(* CODESYS project CtaDevIOMb750362_1.0.0.0.library
   Description: Io System Library für Wago Modbbus Koppler 750-362 der CTA
   Version: 1.0.0.0
   Title: CtaDevIOMb750362
   Author: SIS
   DocFormat: reStructuredText
   LanguageModelAttribute: qualified-access-only
   Placeholder: CtaDevIOMb750362
   CompiledLibraryCompatibilityVersion: CODESYS V3.5 SP16 Patch 3
   Company: CTA
   DefaultNamespace: CtaDevIOMb750362

Project tree, tasks and I/O mapping:
  libraries: Standard, 3.5.18.0 (System); VisuDialogs, * (System); CtaSysConfig, 2.0.0.0 (CTA); CtaAppReport, 2.0.0.0 (CTA); CtaAppBmk, 2.0.0.0 (CTA); CtaAppInfluxLog, 1.0.0.1 (CTA); SysCom, 3.5.17.0 (System); CtaAppModbus, 2.0.0.0 (CTA); CtaSysIO, 2.0.0.0 (CTA); CtaVisSymbols, 2.0.0.0 (CTA)
  40 Visualizations/
    visualisation DIA_MB750362
    PFC_SLOT/
      SLOT/
        visualisation VIS_SLOT
        visualisation VIS_SLOT_QUERY
      FC/
        visualisation VIS_FC
        visualisation VIS_FC_QUERY
      visualisation FC_SLOT
      visualisation FC_SLOT_QUERY
    visualisation IO_ManagerBusInfo
    visualisation VIS_DYN_FC_IO_BASE
  30 Program Organization Units/
    function block FB_MB750362_KOPPLER [ST]: proVISU_DIA_NAME, actReport, BUS_ERROR, SIM_IO_TYPE
    FC/
      function fcScaleOut0_20mA [ST]
      function FcCheckIsDigitalIO [ST]
      function fcScaleOut4_20mA [ST]
      function fcGetTypeOfWagoSlot [ST]
      function fcScaleIN0_20mA [ST]
      function fcScaleOut0_10V [ST]
      function fcScaleIN0_10V [ST]
      function fcScaleIN4_20mA [ST]
      function fcScalePT1000 [ST]
      function fcGetModulImage [ST]
      function fcGetTypeOfWagoSlotSim [ST]
      function FcGetDigitalIOSim [ST]
  00000000-0000-0000-0000-000000000000|D:\CoDeSys\LibrariesV3\trunk\Intern\CAA\CAA Template\3.4.0.0 draft\Placeholder.xml
  00000000-0000-0000-0000-000000000000|D:\CoDeSys\LibrariesV3\trunk\Intern\CAA\CAA Template\3.2.0.3 draft\Prefix.pdf
  00000000-0000-0000-0000-000000000000|D:\CoDeSys\LibrariesV3\trunk\Intern\CAA\CAA Template\3.5.2.0 draft\Placeholder.xml
  20 Structs/
    data type scSlotInfo
    data type enModuleType
  50 Images/
    image pool WAGO_MB_IO_TERMINALS
  10 Documenation/
    global variables VersionHistory
    global variables readMe
  21 Interface/
  11 Library Parameter/
    global variables Parameter
  12 Konstanten/
  60 Textlisten/
    text list txtModulType
    text list txtWarning
    text list txtError
    text list txtPhysicalUnit
    text list txtInfo
  13 Globale Variablen/
    global variables GVL_TEXTLIST
  text list GlobalTextList
  5ce3da45-db07-42e7-a21c-a00fff4ed8f6|S:\_Temporär_SIS\CtaCodesysLibrary\01_Library\CtaSysIO\04_Image\0750_400.bmp
  5ce3da45-db07-42e7-a21c-a00fff4ed8f6|S:\_Temporär_SIS\CtaCodesysLibrary\01_Library\CtaSysIO\04_Image\0750_432.bmp
  5ce3da45-db07-42e7-a21c-a00fff4ed8f6|S:\_Temporär_SIS\CtaCodesysLibrary\01_Library\CtaSysIO\04_Image\0750_451.bmp
  5ce3da45-db07-42e7-a21c-a00fff4ed8f6|S:\_Temporär_SIS\CtaCodesysLibrary\01_Library\CtaSysIO\04_Image\0750_455.bmp
  5ce3da45-db07-42e7-a21c-a00fff4ed8f6|S:\_Temporär_SIS\CtaCodesysLibrary\01_Library\CtaSysIO\04_Image\0750_459.bmp
  5ce3da45-db07-42e7-a21c-a00fff4ed8f6|S:\_Temporär_SIS\CtaCodesysLibrary\01_Library\CtaSysIO\04_Image\0750_466.bmp
  5ce3da45-db07-42e7-a21c-a00fff4ed8f6|S:\_Temporär_SIS\CtaCodesysLibrary\01_Library\CtaSysIO\04_Image\0750_515.bmp
  5ce3da45-db07-42e7-a21c-a00fff4ed8f6|S:\_Temporär_SIS\CtaCodesysLibrary\01_Library\CtaSysIO\04_Image\0750_597.bmp
  5ce3da45-db07-42e7-a21c-a00fff4ed8f6|\\cta.local\mue\Daten\200_Klima_Kälte\200_300_KK_CTA_Exklusiv_Elektro\01_Elektro\03_Software\00_CtaCodesysLibrary\01_Library\CtaDevIOMb750362\04_Image\0750_600.bmp
  5ce3da45-db07-42e7-a21c-a00fff4ed8f6|S:\_Temporär_SIS\CtaCodesysLibrary\01_Library\CtaSysIO\04_Image\0750_652.bmp
  5ce3da45-db07-42e7-a21c-a00fff4ed8f6|S:\_Temporär_SIS\CtaCodesysLibrary\01_Library\CtaSysIO\04_Image\0750_1405.bmp
  5ce3da45-db07-42e7-a21c-a00fff4ed8f6|S:\_Temporär_SIS\CtaCodesysLibrary\01_Library\CtaSysIO\04_Image\0750_1415.bmp
  5ce3da45-db07-42e7-a21c-a00fff4ed8f6|S:\_Temporär_SIS\CtaCodesysLibrary\01_Library\CtaSysIO\04_Image\0750_1504.bmp
  5ce3da45-db07-42e7-a21c-a00fff4ed8f6|P:\200_Klima_Kälte\200_300_KK_CTA_Exklusiv_Elektro\01_Elektro\03_Software\00_CtaCodesysLibrary\01_Library\CtaDevIOMb750362\04_Image\0750_362.png
  5ce3da45-db07-42e7-a21c-a00fff4ed8f6|\\cta.local\mue\Daten\200_Klima_Kälte\200_300_KK_CTA_Exklusiv_Elektro\01_Elektro\03_Software\00_CtaCodesysLibrary\01_Library\CtaDevIOMb750362\04_Image\0750_BLANK.bmp
  5ce3da45-db07-42e7-a21c-a00fff4ed8f6|S:\_Temporär_SIS\CtaCodesysLibrary\01_Library\CtaSysIO\04_Image\0750_555.bmp
*)

// 20 Structs/scSlotInfo
TYPE scSlotInfo :
	STRUCT
		uiOrderNr	:	UINT;
		xDigital	:	BOOL;
		xInput		:	BOOL;
		uiFirstData	:	UINT;
		uiLastData	:	UINT;
		byAnzIoSlot	:	BYTE;
		enModulType :	enModuleType;
	END_STRUCT
END_TYPE

// 20 Structs/enModuleType
{attribute 'qualified_only'}
{attribute 'strict'}
{attribute 'to_string'}
TYPE enModuleType :
(
	Unknown 		:= 0,
	Digital_IN		:= 1,
	Digital_OUT		:= 2,	
	DC_0_10V_OUT	:= 3,
	DC_4_20mA_OUT	:= 4,
	DC_0_10V_IN		:= 5,
	DC_4_20mA_IN	:= 6,
	OHM				:= 7,
    RS485			:= 8,
	DC_0_20mA_OUT	:= 9,
	TEMPERATUR		:= 10,
	FCMB750362		:= 99
);
END_TYPE

// 10 Documenation/VersionHistory
(* 

.. image:: ../../Images/CTA_Logo.jpg
   :align: right
   :width: 15% 

**Vorlage**   


============ =========== =========== ============================================
**Date**     **Version** **Author**  **Change**
------------ ----------- ----------- --------------------------------------------
04.03.2021   0.0.0.0     SIS         Vorlage erstellt

============ =========== =========== ============================================


*)
VAR_GLOBAL
    stInfo : STRING:= '0.0.0.0, Vorlage, CTA';
END_VAR

// 10 Documenation/readMe
(*

**ReadMe**
 
|	**Empfehlung**
|
|	Dokumentrieren Sie die Library für eine nachhaltige Entwicklung
|     
| *Beispiel*
| 
| Dies ist die Vorlage Library der CTA. Erstellen Sie ihre Library anhand dieser Vorlage.
*)

VAR_GLOBAL
    xReadMeDone              :   BOOL;
END_VAR

// 11 Library Parameter/Parameter
{attribute 'qualified_only'}
VAR_GLOBAL CONSTANT

END_VAR

// 13 Globale Variablen/GVL_TEXTLIST
{attribute 'qualified_only'}
VAR_GLOBAL CONSTANT
	stErrorTextlist		:	CtaAppReport.stReportTextList	:= 'CtaDevIOMb750362.txtError';
	stWarningTextlist	:	CtaAppReport.stReportTextList	:= 'CtaDevIOMb750362.txtWarning';
	stInfoTextlist		:	CtaAppReport.stReportTextList	:= 'CtaDevIOMb750362.txtInfo';
END_VAR

// 30 Program Organization Units/FB_MB750362_KOPPLER
FUNCTION_BLOCK FB_MB750362_KOPPLER EXTENDS CtaSysIO.FB_IO_DEVICE
VAR_INPUT
	ITF_CLIENT_IN		:	CtaAppModbus.ITF_CLIENT;
END_VAR
VAR_OUTPUT
	xAcknowledge		:	BOOL;
	xLockDown			:	BOOL;
END_VAR
VAR
	(* Data *)
	_wKbusReset			:	WORD;
	_wSoftWareReset		:	WORD;
	_ayDiagnose			:	ARRAY[0..0001]	OF WORD;
	_ayWatchDog			:	ARRAY[0..0010] 	OF WORD;
	_aySlotType			:	ARRAY[0..0255] 	OF WORD;
	_ayIOQuantity		:	ARRAY[0..0003] 	OF WORD;
	_ayAnalogInput		:	ARRAY[0..1020]	OF WORD;
	_ayAnalogOutput		:	ARRAY[0..1020]	OF WORD;
	_ayDigitalInput		:	ARRAY[0..0511]	OF BOOL;
	_ayDigitalOutput	:	ARRAY[0..0511]	OF BOOL;
	_aySlotInfo			:	ARRAY[0..0255]	OF scSlotInfo;	
	byAnzSlots			:	BYTE;
	(* Help Variable *)
	xTrigResetDevError	:	BOOL;
	xTrigResetSlotError	:	BOOL;
	xReset				:	BOOL;
	usiCase				:	USINT;
	diFor				:	DINT;
	diFor2				:	DINT;	
	diStartFor			:	DINT;
	diMaxCreatePerCycle	:	DINT	:= 50;	
	byAnzIoSlot			:	BYTE;
	uiNextAnalogInput	:	UINT;
	uiNextAnalogOutput	:	UINT;
	uiNextDigitalInput	:	UINT;
	uiNextDigitalOutput :	UINT;
	ITF_SLOT_TEMP		:	CtaSysIO.ITF_IO_SLOT;
	ITF_DI_TEMP			:	CtaSysIO.ITF_DI;
	ITF_DO_TEMP			:	CtaSysIO.ITF_DO;
	ITF_AI_TEMP			:	CtaSysIO.ITF_AI;
	ITF_AO_TEMP			:	CtaSysIO.ITF_AO;
	enType				:	CtaSysIO.enIOType;
	xTempAlUnterlauf	:	BOOL;
	xTempAlUeberlauf	:	BOOL;
	rTempPhysicalValue	:	REAL;
	tErrorDelayMb		:	TIME	:= T#20S;
	xBusError			:	BOOL;
	scReportNr			:	CtaAppReport.scReportNr;
	fbReportManager		:	CtaAppReport.fbReportManager;
	fbMbErrorReport		:	CtaAppReport.fbReporter;
	fbDevErrorReport	:	CtaAppReport.fbReporter;
	fbWarningReportHand	:	CtaAppReport.fbReporter;
	fbSlotMissmatch		:	CtaAppReport.fbReporter;
END_VAR;

SUPER^();
IF NOT SIMULATION_ENABLED THEN
	IF __QUERYINTERFACE(ITF_CLIENT_IN,ITF_CLIENT_IN) THEN
		xBusError := ITF_CLIENT_IN.ERROR;
		CASE usiCase OF 
			0:  (* Set Image *)
				IMAGE := '.WAGO_MB_IO_TERMINALS.0750_362';
				(* Read Watchdog State *)
				ITF_CLIENT_IN.CREATE_JOB(_byMbFunction := 04,_wMbAdress := 4102,_pData := ADR(_ayWatchDog[006])	,_wQuantity := 01);
				
				(* Reset K-Bus *)
				ITF_CLIENT_IN.CREATE_JOB(_byMbFunction := 06,_wMbAdress := 4139,_pData := ADR(_wKbusReset)		,_wQuantity := 01);
	
				(* Diagnose Info *)
				ITF_CLIENT_IN.CREATE_JOB(_byMbFunction := 04,_wMbAdress := 4128,_pData := ADR(_ayDiagnose[000])	,_wQuantity := 2);
				
				(* Next Step *)
				usiCase := usiCase + 1;
				
			1:	(* Wait *)
				IF ITF_CLIENT_IN.CONFIRM_ALL_JOBS_DONE THEN
					(* Next Step *)
					usiCase := usiCase + 1;
				END_IF;
				
			2:	(* Watchdog State evaluvation *)
				IF _ayWatchDog[06] = 0 THEN // Watchdog inaktive
					(* Set Watchdog Time *)
					_ayWatchDog[00]	:= 16#0032;	// Watchdog Time 5s
					ITF_CLIENT_IN.CREATE_JOB(_byMbFunction := 06,_wMbAdress := 4096,_pData := ADR(_ayWatchDog[000])	,_wQuantity := 01);
					(* Set Watchdog Reset Funktion *)
					_ayWatchDog[01]	:= 16#FFFF;	// Reset on FC1-FC16
					ITF_CLIENT_IN.CREATE_JOB(_byMbFunction := 06,_wMbAdress := 4097,_pData := ADR(_ayWatchDog[001])	,_wQuantity := 01);
					(* Remove Watchdog Stop Call *)
					ITF_CLIENT_IN.DESTROY_JOB(_byMbFunction := 06,_wMbAdress := 4104,_pData := ADR(_ayWatchDog[008])	,_wQuantity := 01);
					(* Remove K-Bus reset *)
					ITF_CLIENT_IN.DESTROY_JOB(_byMbFunction := 06,_wMbAdress := 4139,_pData := ADR(_wKbusReset)		,_wQuantity := 01);
					(* Remove Software reset *)
					ITF_CLIENT_IN.DESTROY_JOB(_byMbFunction := 06,_wMbAdress :=8256,_pData 	:=	 ADR(_wSoftWareReset),	_wQuantity	 :=	 1);
					(* Next Step after Watchdog Set *)
					usiCase := usiCase + 1;
				(* Stop Watchdog if allredy aktive *)
				ELSIF _ayWatchDog[06] = 1 OR _ayWatchDog[06] = 2 THEN // Watchdog aktive or Watchdog expired
					_ayWatchDog[08]	:= 16#AA55;	// Watchdog Stop
					ITF_CLIENT_IN.CREATE_JOB(_byMbFunction := 06,_wMbAdress := 4104,_pData := ADR(_ayWatchDog[008])	,_wQuantity := 01); 
				END_IF;
				
			3:	(* Wait *)
				IF ITF_CLIENT_IN.CONFIRM_ALL_JOBS_DONE THEN
					(* Next Step *)
					usiCase := usiCase + 1;
				END_IF;
				
			4: (* Check if Watchdog is Running *)
					(* Read Slots *)
					ITF_CLIENT_IN.CREATE_JOB(_byMbFunction 	:= 04,	_wMbAdress 	:= 8240,	_pData 	:=	 ADR(_aySlotType[000]),	_wQuantity	 :=	 65);
					ITF_CLIENT_IN.CREATE_JOB(_byMbFunction 	:= 04,	_wMbAdress 	:= 8241,	_pData 	:=	 ADR(_aySlotType[065]),	_wQuantity	 :=	 64);
					ITF_CLIENT_IN.CREATE_JOB(_byMbFunction 	:= 04,	_wMbAdress 	:= 8242,	_pData 	:=	 ADR(_aySlotType[129]),	_wQuantity	 :=	 64);
					ITF_CLIENT_IN.CREATE_JOB(_byMbFunction 	:= 04,	_wMbAdress 	:= 8243,	_pData 	:=	 ADR(_aySlotType[193]),	_wQuantity	 :=	 63);	
					
					(* Read Quantity of I/O *)                                          	       	  	                                  	   	
					ITF_CLIENT_IN.CREATE_JOB(_byMbFunction 	:= 04,	_wMbAdress 	:= 4130,	_pData 	:=	 ADR(_ayIOQuantity[0]),	_wQuantity	 :=	 04);	
				IF _ayWatchDog[06] = 1 THEN	
					(* Remove Watchdog Configs *)                                       	       	  	                                  	   	
					ITF_CLIENT_IN.DESTROY_JOB(_byMbFunction := 06,	_wMbAdress 	:= 4096,	_pData 	:=	 ADR(_ayWatchDog[000]),	_wQuantity	 :=	 01);
					ITF_CLIENT_IN.DESTROY_JOB(_byMbFunction := 06,	_wMbAdress 	:= 4097,	_pData 	:=	 ADR(_ayWatchDog[001]),	_wQuantity	 :=	 01);
					
					(* Next Step *)
					usiCase := usiCase + 1;                                             	       	  	                                       	
				END_IF;    
																														
			5:	(* Wait *)                                                              	       	  	                                       	
				IF ITF_CLIENT_IN.CONFIRM_ALL_JOBS_DONE THEN 
					(* Next Step *)                            	       	  	                                       	
					usiCase := usiCase + 1;                                             	       	  	                                       	
				END_IF;	
																															
			6: 	(* Delete Slot Jobs *)                                                  	       	  	                                       	
				ITF_CLIENT_IN.DESTROY_JOB(_byMbFunction 	:= 04,	_wMbAdress 	:= 8240,	_pData 	:=	 ADR(_aySlotType[000]),	_wQuantity	 :=	 65);
				ITF_CLIENT_IN.DESTROY_JOB(_byMbFunction 	:= 04,	_wMbAdress 	:= 8241,	_pData 	:=	 ADR(_aySlotType[065]),	_wQuantity	 :=	 64);
				ITF_CLIENT_IN.DESTROY_JOB(_byMbFunction 	:= 04,	_wMbAdress 	:= 8242,	_pData 	:=	 ADR(_aySlotType[129]),	_wQuantity	 :=	 64);
				ITF_CLIENT_IN.DESTROY_JOB(_byMbFunction 	:= 04,	_wMbAdress 	:= 8243,	_pData 	:=	 ADR(_aySlotType[193]),	_wQuantity	 :=	 63);	
				
				(* Delte Quantity of I/O *)                                             	       	  	                                  	   	
				ITF_CLIENT_IN.DESTROY_JOB(_byMbFunction 	:= 04,	_wMbAdress 	:= 4130,	_pData 	:=	 ADR(_ayIOQuantity[0]),	_wQuantity	 :=	 04);
				
				(* Add Read Analog Input Jobs as needed *)  
				IF (_ayIOQuantity[1] / 16) >= 001 THEN   // Quantity is Bit Orientet /16 = Dezimal                                           	       	  	                                  	   	
					ITF_CLIENT_IN.CREATE_JOB(_byMbFunction 		:= 04,	_wMbAdress 	:= 0000,	_pData 	:=	 ADR(_ayAnalogInput[000]),	_wQuantity	 :=	 MAX(1,MIN(085,(_ayIOQuantity[1] / 16) -000)));
				END_IF;
				IF (_ayIOQuantity[1] / 16) >= 085 THEN   // Quantity is Bit Orientet /16 = Dezimal 
					ITF_CLIENT_IN.CREATE_JOB(_byMbFunction 		:= 04,	_wMbAdress 	:= 0085,	_pData 	:=	 ADR(_ayAnalogInput[085]),	_wQuantity	 :=	 MAX(1,MIN(085,(_ayIOQuantity[1] / 16) -085)));
				END_IF;
				IF (_ayIOQuantity[1] / 16) >= 170 THEN   // Quantity is Bit Orientet /16 = Dezimal 
					ITF_CLIENT_IN.CREATE_JOB(_byMbFunction 		:= 04,	_wMbAdress 	:= 0170,	_pData 	:=	 ADR(_ayAnalogInput[170]),	_wQuantity	 :=	 MAX(1,MIN(086,(_ayIOQuantity[1] / 16) -170)));
				END_IF;
				IF (_ayIOQuantity[1] / 16) >= 256 THEN   // Quantity is Bit Orientet /16 = Dezimal 
					ITF_CLIENT_IN.CREATE_JOB(_byMbFunction 		:= 04,	_wMbAdress 	:=24576,	_pData 	:=	 ADR(_ayAnalogInput[256]),	_wQuantity	 :=	 MAX(1,MIN(120,(_ayIOQuantity[1] / 16) -256)));
				END_IF;
				IF (_ayIOQuantity[1] / 16) >= 376 THEN   // Quantity is Bit Orientet /16 = Dezimal 
					ITF_CLIENT_IN.CREATE_JOB(_byMbFunction 		:= 04,	_wMbAdress 	:=24696,	_pData 	:=	 ADR(_ayAnalogInput[376]),	_wQuantity	 :=	 MAX(1,MIN(120,(_ayIOQuantity[1] / 16) -376)));
				END_IF;
				IF (_ayIOQuantity[1] / 16) >= 496 THEN   // Quantity is Bit Orientet /16 = Dezimal 
					ITF_CLIENT_IN.CREATE_JOB(_byMbFunction 		:= 04,	_wMbAdress 	:=24816,	_pData 	:=	 ADR(_ayAnalogInput[496]),	_wQuantity	 :=	 MAX(1,MIN(120,(_ayIOQuantity[1] / 16) -496)));
				END_IF;
				IF (_ayIOQuantity[1] / 16) >= 616 THEN   // Quantity is Bit Orientet /16 = Dezimal 
					ITF_CLIENT_IN.CREATE_JOB(_byMbFunction 		:= 04,	_wMbAdress 	:=24936,	_pData 	:=	 ADR(_ayAnalogInput[616]),	_wQuantity	 :=	 MAX(1,MIN(120,(_ayIOQuantity[1] / 16) -616)));
				END_IF;
				IF (_ayIOQuantity[1] / 16) >= 736 THEN   // Quantity is Bit Orientet /16 = Dezimal 
					ITF_CLIENT_IN.CREATE_JOB(_byMbFunction 		:= 04,	_wMbAdress 	:=25056,	_pData 	:=	 ADR(_ayAnalogInput[736]),	_wQuantity	 :=	 MAX(1,MIN(120,(_ayIOQuantity[1] / 16) -736)));
				END_IF;
				IF (_ayIOQuantity[1] / 16) >= 856 THEN   // Quantity is Bit Orientet /16 = Dezimal 
					ITF_CLIENT_IN.CREATE_JOB(_byMbFunction 		:= 04,	_wMbAdress 	:=25176,	_pData 	:=	 ADR(_ayAnalogInput[856]),	_wQuantity	 :=	 MAX(1,MIN(120,(_ayIOQuantity[1] / 16) -856)));
				END_IF;
				IF (_ayIOQuantity[1] / 16) >= 976 THEN   // Quantity is Bit Orientet /16 = Dezimal 
					ITF_CLIENT_IN.CREATE_JOB(_byMbFunction 		:= 04,	_wMbAdress 	:=25296,	_pData 	:=	 ADR(_ayAnalogInput[976]),	_wQuantity	 :=	 MAX(1,MIN(044,(_ayIOQuantity[1] / 16) -976)));
				END_IF;
				
				(* Add Write Analog Output Jobs *)      
				IF (_ayIOQuantity[0] / 16) >= 001 THEN   // Quantity is Bit Orientet /16 = Dezimal                                                                        	       	  	                                  	   	
					ITF_CLIENT_IN.CREATE_JOB(_byMbFunction 		:= 16,	_wMbAdress 	:= 0000,	_pData 	:=	 ADR(_ayAnalogOutput[000]),	_wQuantity	 :=	 MAX(1,MIN(085,(_ayIOQuantity[0] / 16) -000)));
				END_IF;                                                                                                                                                                                
				IF (_ayIOQuantity[0] / 16) >= 085  THEN   // Quantity is Bit Orientet /16 = Dezimal                                                                                                    
					ITF_CLIENT_IN.CREATE_JOB(_byMbFunction 		:= 16,	_wMbAdress 	:= 0085,	_pData 	:=	 ADR(_ayAnalogOutput[085]),	_wQuantity	 :=	 MAX(1,MIN(085,(_ayIOQuantity[0] / 16) -085)));
				END_IF;                                                                                                                                                                                
				IF (_ayIOQuantity[0] / 16) >= 170  THEN   // Quantity is Bit Orientet /16 = Dezimal                                                                                                    
					ITF_CLIENT_IN.CREATE_JOB(_byMbFunction 		:= 16,	_wMbAdress 	:= 0170,	_pData 	:=	 ADR(_ayAnalogOutput[170]),	_wQuantity	 :=	 MAX(1,MIN(086,(_ayIOQuantity[0] / 16) -170)));
				END_IF;                                                                                                                                                                                
				IF (_ayIOQuantity[0] / 16) >= 256  THEN   // Quantity is Bit Orientet /16 = Dezimal                                                                                                    
					ITF_CLIENT_IN.CREATE_JOB(_byMbFunction 		:= 16,	_wMbAdress 	:=24576,	_pData 	:=	 ADR(_ayAnalogOutput[256]),	_wQuantity	 :=	 MAX(1,MIN(120,(_ayIOQuantity[0] / 16) -256)));
				END_IF;                                                                                                                                                                                
				IF (_ayIOQuantity[0] / 16) >= 376 THEN   // Quantity is Bit Orientet /16 = Dezimal                                                                                                     
					ITF_CLIENT_IN.CREATE_JOB(_byMbFunction 		:= 16,	_wMbAdress 	:=24696,	_pData 	:=	 ADR(_ayAnalogOutput[376]),	_wQuantity	 :=	 MAX(1,MIN(120,(_ayIOQuantity[0] / 16) -376)));
				END_IF;                                                                                                                                                                                
				IF (_ayIOQuantity[0] / 16) >= 496 THEN   // Quantity is Bit Orientet /16 = Dezimal                                                                                                     
					ITF_CLIENT_IN.CREATE_JOB(_byMbFunction 		:= 16,	_wMbAdress 	:=24816,	_pData 	:=	 ADR(_ayAnalogOutput[496]),	_wQuantity	 :=	 MAX(1,MIN(120,(_ayIOQuantity[0] / 16) -496)));
				END_IF;                                                                                                                                                                                
				IF (_ayIOQuantity[0] / 16) >= 616 THEN   // Quantity is Bit Orientet /16 = Dezimal                                                                                                     
					ITF_CLIENT_IN.CREATE_JOB(_byMbFunction 		:= 16,	_wMbAdress 	:=24936,	_pData 	:=	 ADR(_ayAnalogOutput[616]),	_wQuantity	 :=	 MAX(1,MIN(120,(_ayIOQuantity[0] / 16) -616)));
				END_IF;                                                                                                                                                                                
				IF (_ayIOQuantity[0] / 16) >= 736 THEN   // Quantity is Bit Orientet /16 = Dezimal                                                                                                     
					ITF_CLIENT_IN.CREATE_JOB(_byMbFunction 		:= 16,	_wMbAdress 	:=25056,	_pData 	:=	 ADR(_ayAnalogOutput[736]),	_wQuantity	 :=	 MAX(1,MIN(120,(_ayIOQuantity[0] / 16) -736)));
				END_IF;                                                                                                                                                                                
				IF (_ayIOQuantity[0] / 16) >= 856 THEN   // Quantity is Bit Orientet /16 = Dezimal                                                                                                     
					ITF_CLIENT_IN.CREATE_JOB(_byMbFunction 		:= 16,	_wMbAdress 	:=25176,	_pData 	:=	 ADR(_ayAnalogOutput[856]),	_wQuantity	 :=	 MAX(1,MIN(120,(_ayIOQuantity[0] / 16) -856)));
				END_IF;                                                                                                                                                                                
				IF (_ayIOQuantity[0] / 16) >= 976 THEN   // Quantity is Bit Orientet /16 = Dezimal                                                                                                     
					ITF_CLIENT_IN.CREATE_JOB(_byMbFunction 		:= 16,	_wMbAdress 	:=25296,	_pData 	:=	 ADR(_ayAnalogOutput[976]),	_wQuantity	 :=	 MAX(1,MIN(044,(_ayIOQuantity[0] / 16) -976)));
				END_IF;                                                                                                                                  
				
				(* Add Read Digital Input Jobs *)                                                  	       	  	                                  	   	
				ITF_CLIENT_IN.CREATE_JOB(_byMbFunction 		:= 02,	_wMbAdress 	:= 0000,	_pData 	:=	 ADR(_ayDigitalInput[000]),	_wQuantity	 :=	 512);	
		
				(* Add Read Digital Input Jobs *)                                                  	       	  	                                  	   	
				ITF_CLIENT_IN.CREATE_JOB(_byMbFunction 		:= 15,	_wMbAdress 	:= 0000,	_pData 	:=	 ADR(_ayDigitalOutput[000]),_wQuantity	 :=	 512);		
		
				usiCase := usiCase + 1;
			7:	(* Wait *)
				IF ITF_CLIENT_IN.CONFIRM_ALL_JOBS_DONE THEN
					(* Reset IO State *)
					uiNextAnalogInput	:= 0;
					uiNextAnalogOutput	:= 0;
					uiNextDigitalInput	:= 0;
					uiNextDigitalOutput := 0;
					FOR diFor := LOWER_BOUND(_aySlotInfo,1) TO UPPER_BOUND(_aySlotInfo,1) DO
						_aySlotInfo[diFor].uiOrderNr 	:= 0;
						_aySlotInfo[diFor].enModulType 	:= enModuleType.Unknown;
						_aySlotInfo[diFor].xInput		:= FALSE;
						_aySlotInfo[diFor].xDigital		:= FALSE;
						_aySlotInfo[diFor].uiFirstData	:= 0;
						_aySlotInfo[diFor].uiLastData	:= 0;
					END_FOR;
					(* Next Step *) 
					usiCase := usiCase + 1;
				END_IF;
			8: (* Calculate IO *)	
				FOR diFor := LOWER_BOUND(_aySlotType,1) TO UPPER_BOUND(_aySlotType,1) DO
					(* Check if Slot is used *)
					IF _aySlotType[diFor] <> 0 THEN
						(* Count *)
						byAnzSlots	:= TO_BYTE(diFor);
						(* Check if Valid Info array *)
						IF diFor >= LOWER_BOUND(_aySlotInfo,1) AND diFor <= UPPER_BOUND(_aySlotInfo,1) THEN
							(* Get Type of Slot *)
							_aySlotInfo[diFor].uiOrderNr := fcGetTypeOfWagoSlot(wInput := _aySlotType[difor],xIsInput => _aySlotInfo[diFor].xInput, xIsDigital => _aySlotInfo[diFor].xDigital,byAnzIo => byAnzIoSlot,enModulType =>_aySlotInfo[diFor].enModulType);
							IF byAnzIoSlot > 0 THEN
								(* Anzahl IO *)
								_aySlotInfo[diFor].byAnzIoSlot := byAnzIoSlot;
								(* Digital *)
								IF _aySlotInfo[diFor].xDigital THEN
									(* Input *)
									IF _aySlotInfo[diFor].xInput THEN
										_aySlotInfo[diFor].uiFirstData 	:= uiNextDigitalInput;
										_aySlotInfo[diFor].uiLastData	:= uiNextDigitalInput + byAnzIoSlot - 1;	// -1 because of 0 based start
										uiNextDigitalInput := uiNextDigitalInput + byAnzIoSlot;
									(* Output *)
									ELSE
										_aySlotInfo[diFor].uiFirstData 	:= uiNextDigitalOutput;
										_aySlotInfo[diFor].uiLastData	:= uiNextDigitalOutput + byAnzIoSlot - 1;	// -1 because of 0 based start
										uiNextDigitalOutput := uiNextDigitalOutput + byAnzIoSlot;		
									END_IF;
								(* Analog *)
								ELSE
									(* Input *)
									IF _aySlotInfo[diFor].xInput THEN
										_aySlotInfo[diFor].uiFirstData 	:= uiNextAnalogInput;
										_aySlotInfo[diFor].uiLastData	:= uiNextAnalogInput + byAnzIoSlot - 1;	// -1 because of 0 based start
										uiNextAnalogInput := uiNextAnalogInput + byAnzIoSlot;
									(* Output *)
									ELSE
										_aySlotInfo[diFor].uiFirstData 	:= uiNextAnalogOutput;
										_aySlotInfo[diFor].uiLastData	:= uiNextAnalogOutput + byAnzIoSlot - 1;	// -1 because of 0 based start
										uiNextAnalogOutput := uiNextAnalogOutput + byAnzIoSlot;		
									END_IF							
								END_IF
							END_IF;
						END_IF;
					ELSE
						EXIT;
					END_IF;
				END_FOR;
				
				(* Next Step *) 
				usiCase := usiCase + 1;		
				
			9: (* Create I/Os *)
				IF diStartFor = 0 THEN
					diStartFor := LOWER_BOUND(_aySlotInfo,1);
				END_IF
				IF diStartFor <= TO_DINT(byAnzSlots) AND TO_DINT(byAnzSlots) > 0 THEN
					FOR diFor := diStartFor TO TO_DINT(byAnzSlots) DO
						IF _aySlotInfo[diFor].byAnzIoSlot > 0 THEN
							FOR diFor2 := 1 TO TO_DINT(_aySlotInfo[diFor].byAnzIoSlot) DO
								CREATE_SLOT(_usiSlotNr := TO_USINT(diFor),_stSlotImage := fcGetModulImage(_aySlotInfo[diFor].uiOrderNr));
								IF __QUERYINTERFACE(GET_SLOT(TO_USINT(diFor)),ITF_SLOT_TEMP) THEN
									IF _aySlotInfo[diFor].enModulType = enModuleType.Digital_IN THEN
										enType := CtaSysIO.enIOType.Digital_IN;
									ELSIF _aySlotInfo[diFor].enModulType = enModuleType.Digital_OUT THEN
										enType := CtaSysIO.enIOType.Digital_OUT;
									ELSIF _aySlotInfo[diFor].enModulType = enModuleType.DC_0_10V_IN THEN
										enType := CtaSysIO.enIOType.DC_0_10V_IN;
									ELSIF _aySlotInfo[diFor].enModulType = enModuleType.DC_4_20mA_IN THEN
										enType := CtaSysIO.enIOType.DC_4_20mA_IN;
									ELSIF _aySlotInfo[diFor].enModulType = enModuleType.TEMPERATUR THEN
										enType := CtaSysIO.enIOType.TEMPERATUR;
									ELSIF _aySlotInfo[diFor].enModulType = enModuleType.DC_0_10V_OUT THEN
										enType := CtaSysIO.enIOType.DC_0_10V_OUT;
									ELSIF _aySlotInfo[diFor].enModulType = enModuleType.DC_0_20mA_OUT THEN
										enType := CtaSysIO.enIOType.DC_0_20mA_OUT;
									ELSIF _aySlotInfo[diFor].enModulType = enModuleType.DC_4_20mA_OUT THEN
										enType := CtaSysIO.enIOType.DC_4_20mA_OUT;
									END_IF;
									ITF_SLOT_TEMP.CREATE_IO(TO_USINT(diFor2),enType);
								END_IF;
							END_FOR;
						END_IF;	
						IF diFor = TO_DINT(byAnzSlots) THEN
							(* END MODUL *)
							CREATE_SLOT(_usiSlotNr := TO_USINT(diFor + 1),_stSlotImage := '.WAGO_MB_IO_TERMINALS.0750_600');
							SET_STATE_READY_TO_SET_CONFIG := TRUE;
							(* Next Step *) 
							usiCase := usiCase + 1;	
						ELSIF diFor = diStartFor + diMaxCreatePerCycle THEN
							diStartFor := diFor + 1;
							EXIT;
						END_IF;
					END_FOR;
				ELSE
					(* Next Step *) 
					usiCase := usiCase + 1;	
					SET_STATE_READY_TO_SET_CONFIG := TRUE;
				END_IF;
				
			10: (* I/O Init done *)
				(* Check Watchdog and Device Error Cyclic *)
				SET_STATE_READY_TO_SET_CONFIG := FALSE;
				IF _ayWatchDog[06] = 2 OR _ayDiagnose[0] > 0 OR xBusError THEN // Watchdog expired or Error
					ADD_ERROR();
					xLockDown	:= TRUE;
					usiCase := usiCase + 1;
				ELSE
					xLockDown	:= xError;	// Error of Supper Block
				END_IF; 
				(* IO Update *)
				FOR diFor := LOWER_BOUND(_aySlotInfo,1) TO TO_DINT(byAnzSlots) DO
					IF _aySlotInfo[diFor].byAnzIoSlot > 0 THEN
						FOR diFor2 := 1 TO TO_DINT(_aySlotInfo[diFor].byAnzIoSlot) DO
							IF __QUERYINTERFACE(GET_SLOT(TO_USINT(diFor)),ITF_SLOT_TEMP) THEN
								(* Digital Input *)
								IF _aySlotInfo[diFor].enModulType = enModuleType.Digital_IN THEN
									enType := CtaSysIO.enIOType.Digital_IN;
									IF __QUERYINTERFACE((ITF_SLOT_TEMP.GET_IO(TO_USINT(diFOr2))),ITF_DI_TEMP) THEN
										ITF_DI_TEMP.metCyclicIoUpdate(	_xChannelIn		:= _ayDigitalInput[_aySlotInfo[diFor].uiFirstData + TO_UINT(diFor2) -1],
																		_xOk 			:= NOT xLockDown);
									END_IF;
								(* Digital Output *)
								ELSIF _aySlotInfo[diFor].enModulType = enModuleType.Digital_OUT THEN
									enType := CtaSysIO.enIOType.Digital_OUT;
									IF __QUERYINTERFACE((ITF_SLOT_TEMP.GET_IO(TO_USINT(diFOr2))),ITF_DO_TEMP) THEN
										ITF_DO_TEMP.metCyclicIoUpdate(	_xChannelOut	=> _ayDigitalOutput[_aySlotInfo[diFor].uiFirstData + TO_UINT(diFor2) -1],
																		_xOk 			:= NOT xLockDown);
									END_IF;
								(* Analog Input 0-10V *)
								ELSIF _aySlotInfo[diFor].enModulType = enModuleType.DC_0_10V_IN THEN
									enType := CtaSysIO.enIOType.DC_0_10V_IN;
									IF __QUERYINTERFACE((ITF_SLOT_TEMP.GET_IO(TO_USINT(diFOr2))),ITF_AI_TEMP) THEN
										ITF_AI_TEMP.metCyclicIoUpdate(	_rPhysicalValue := fcScaleIN0_10V(	wChanelInput :=_ayAnalogInput[_aySlotInfo[diFor].uiFirstData + TO_UINT(diFor2) -1],
																											xAlUnterlauf => xTempAlUnterlauf,
																											xAlUeberlauf => xTempAlUeberlauf),							
																		_xAlUeberlauf 	:= xTempAlUeberlauf, 
																		_xAlUnterlauf 	:= xTempAlUnterlauf,
																		_xOk 			:= NOT xLockDown);
									END_IF
								(* Analog Input 4-20mA *)
								ELSIF _aySlotInfo[diFor].enModulType = enModuleType.DC_4_20mA_IN THEN
									enType := CtaSysIO.enIOType.DC_4_20mA_IN;
									IF __QUERYINTERFACE((ITF_SLOT_TEMP.GET_IO(TO_USINT(diFOr2))),ITF_AI_TEMP) THEN
										ITF_AI_TEMP.metCyclicIoUpdate(	_rPhysicalValue := fcScaleIN4_20mA(	wChanelInput :=_ayAnalogInput[_aySlotInfo[diFor].uiFirstData + TO_UINT(diFor2) -1],
																											xAlUnterlauf => xTempAlUnterlauf,
																											xAlUeberlauf => xTempAlUeberlauf),							
																		_xAlUeberlauf 	:= xTempAlUeberlauf, 
																		_xAlUnterlauf 	:= xTempAlUnterlauf,
																		_xOk 			:= NOT xLockDown);
									END_IF
								(* Analog Input Temperatur *)
								ELSIF _aySlotInfo[diFor].enModulType = enModuleType.TEMPERATUR THEN
									enType := CtaSysIO.enIOType.TEMPERATUR;
									IF __QUERYINTERFACE((ITF_SLOT_TEMP.GET_IO(TO_USINT(diFOr2))),ITF_AI_TEMP) THEN
										ITF_AI_TEMP.metCyclicIoUpdate(	_rPhysicalValue := fcScalePT1000(	wChanelInput :=_ayAnalogInput[_aySlotInfo[diFor].uiFirstData + TO_UINT(diFor2) -1],
																											xAlUnterlauf => xTempAlUnterlauf,
																											xAlUeberlauf => xTempAlUeberlauf),							
																		_xAlUeberlauf 	:= xTempAlUeberlauf, 
																		_xAlUnterlauf 	:= xTempAlUnterlauf,
																		_xOk 			:= NOT xLockDown);
									END_IF
								(* Analog Output 0-10V *)
								ELSIF _aySlotInfo[diFor].enModulType = enModuleType.DC_0_10V_OUT THEN
									enType := CtaSysIO.enIOType.DC_0_10V_OUT;
									IF __QUERYINTERFACE((ITF_SLOT_TEMP.GET_IO(TO_USINT(diFOr2))),ITF_AO_TEMP) THEN
										ITF_AO_TEMP.metCyclicIoUpdate(_rPhysicalValue => rTempPhysicalValue,_xOk := NOT xLockDown);
										_ayAnalogOutput[_aySlotInfo[diFor].uiFirstData + TO_UINT(diFor2) -1] := fcScaleOut0_10V(rTempPhysicalValue);
									END_IF
								(* Analog Output 0-20mA *)
								ELSIF _aySlotInfo[diFor].enModulType = enModuleType.DC_0_20mA_OUT THEN
									enType := CtaSysIO.enIOType.DC_0_20mA_OUT;
									IF __QUERYINTERFACE((ITF_SLOT_TEMP.GET_IO(TO_USINT(diFOr2))),ITF_AO_TEMP) THEN
										ITF_AO_TEMP.metCyclicIoUpdate(_rPhysicalValue => rTempPhysicalValue,_xOk := NOT xLockDown);
										_ayAnalogOutput[_aySlotInfo[diFor].uiFirstData + TO_UINT(diFor2) -1] := fcScaleOut0_20mA(rTempPhysicalValue);
									END_IF
								(* Analog Output 4-20mA *)
								ELSIF _aySlotInfo[diFor].enModulType = enModuleType.DC_4_20mA_OUT THEN
									enType := CtaSysIO.enIOType.DC_4_20mA_OUT;
									IF __QUERYINTERFACE((ITF_SLOT_TEMP.GET_IO(TO_USINT(diFOr2))),ITF_AO_TEMP) THEN
										ITF_AO_TEMP.metCyclicIoUpdate(_rPhysicalValue => rTempPhysicalValue,_xOk := NOT xLockDown);
										_ayAnalogOutput[_aySlotInfo[diFor].uiFirstData + TO_UINT(diFor2) -1] := fcScaleOut4_20mA(rTempPhysicalValue);
									END_IF
								END_IF;
							END_IF;
						END_FOR;
					END_IF;	
				END_FOR;	
				CONFIG_DONE := TRUE;      
				tErrorDelayMb := T#2S;                            	       	  	                                       				
			11: (* On Error destroy all Modbus jobs to garant an Watchdogexeption on the Modbus Device after wait to Reset *)
	
				(* Delete Watchdog State *)
				ITF_CLIENT_IN.DESTROY_JOB(_byMbFunction := 04,_wMbAdress := 4102,_pData := ADR(_ayWatchDog[006])	,_wQuantity := 01);
				
				(* Delete Info *)
				ITF_CLIENT_IN.DESTROY_JOB(_byMbFunction := 04,_wMbAdress := 4128,_pData := ADR(_ayDiagnose[000])	,_wQuantity := 2);		
				
				(* Delete Read Analog Input Jobs *)  
				ITF_CLIENT_IN.DESTROY_JOB(_byMbFunction 		:= 04,	_wMbAdress 	:= 0000,	_pData 	:=	 ADR(_ayAnalogInput[000]),	_wQuantity	 :=	 MAX(1,MIN(085,(_ayIOQuantity[1] / 16) -000)));
				ITF_CLIENT_IN.DESTROY_JOB(_byMbFunction 		:= 04,	_wMbAdress 	:= 0085,	_pData 	:=	 ADR(_ayAnalogInput[085]),	_wQuantity	 :=	 MAX(1,MIN(085,(_ayIOQuantity[1] / 16) -085)));
				ITF_CLIENT_IN.DESTROY_JOB(_byMbFunction 		:= 04,	_wMbAdress 	:= 0170,	_pData 	:=	 ADR(_ayAnalogInput[170]),	_wQuantity	 :=	 MAX(1,MIN(086,(_ayIOQuantity[1] / 16) -170)));
				ITF_CLIENT_IN.DESTROY_JOB(_byMbFunction 		:= 04,	_wMbAdress 	:=24576,	_pData 	:=	 ADR(_ayAnalogInput[256]),	_wQuantity	 :=	 MAX(1,MIN(120,(_ayIOQuantity[1] / 16) -256)));
				ITF_CLIENT_IN.DESTROY_JOB(_byMbFunction 		:= 04,	_wMbAdress 	:=24696,	_pData 	:=	 ADR(_ayAnalogInput[376]),	_wQuantity	 :=	 MAX(1,MIN(120,(_ayIOQuantity[1] / 16) -376)));
				ITF_CLIENT_IN.DESTROY_JOB(_byMbFunction 		:= 04,	_wMbAdress 	:=24816,	_pData 	:=	 ADR(_ayAnalogInput[496]),	_wQuantity	 :=	 MAX(1,MIN(120,(_ayIOQuantity[0] / 16) -496)));
				ITF_CLIENT_IN.DESTROY_JOB(_byMbFunction 		:= 04,	_wMbAdress 	:=24936,	_pData 	:=	 ADR(_ayAnalogInput[616]),	_wQuantity	 :=	 MAX(1,MIN(120,(_ayIOQuantity[1] / 16) -616)));
				ITF_CLIENT_IN.DESTROY_JOB(_byMbFunction 		:= 04,	_wMbAdress 	:=25056,	_pData 	:=	 ADR(_ayAnalogInput[736]),	_wQuantity	 :=	 MAX(1,MIN(120,(_ayIOQuantity[1] / 16) -736)));
				ITF_CLIENT_IN.DESTROY_JOB(_byMbFunction 		:= 04,	_wMbAdress 	:=25176,	_pData 	:=	 ADR(_ayAnalogInput[856]),	_wQuantity	 :=	 MAX(1,MIN(120,(_ayIOQuantity[1] / 16) -856)));
				ITF_CLIENT_IN.DESTROY_JOB(_byMbFunction 		:= 04,	_wMbAdress 	:=25296,	_pData 	:=	 ADR(_ayAnalogInput[976]),	_wQuantity	 :=	 MAX(1,MIN(044,(_ayIOQuantity[1] / 16) -976)));
				
				(* Delete Write Analog Output Jobs *)      
				ITF_CLIENT_IN.DESTROY_JOB(_byMbFunction 		:= 16,	_wMbAdress 	:= 0000,	_pData 	:=	 ADR(_ayAnalogOutput[000]),	_wQuantity	 :=	 MAX(1,MIN(085,(_ayIOQuantity[0] / 16) -000)));
				ITF_CLIENT_IN.DESTROY_JOB(_byMbFunction 		:= 16,	_wMbAdress 	:= 0085,	_pData 	:=	 ADR(_ayAnalogOutput[085]),	_wQuantity	 :=	 MAX(1,MIN(085,(_ayIOQuantity[0] / 16) -085)));
				ITF_CLIENT_IN.DESTROY_JOB(_byMbFunction 		:= 16,	_wMbAdress 	:= 0170,	_pData 	:=	 ADR(_ayAnalogOutput[170]),	_wQuantity	 :=	 MAX(1,MIN(086,(_ayIOQuantity[0] / 16) -170)));
				ITF_CLIENT_IN.DESTROY_JOB(_byMbFunction 		:= 16,	_wMbAdress 	:=24576,	_pData 	:=	 ADR(_ayAnalogOutput[256]),	_wQuantity	 :=	 MAX(1,MIN(120,(_ayIOQuantity[0] / 16) -256)));
				ITF_CLIENT_IN.DESTROY_JOB(_byMbFunction 		:= 16,	_wMbAdress 	:=24696,	_pData 	:=	 ADR(_ayAnalogOutput[376]),	_wQuantity	 :=	 MAX(1,MIN(120,(_ayIOQuantity[0] / 16) -376)));
				ITF_CLIENT_IN.DESTROY_JOB(_byMbFunction 		:= 16,	_wMbAdress 	:=24816,	_pData 	:=	 ADR(_ayAnalogOutput[496]),	_wQuantity	 :=	 MAX(1,MIN(120,(_ayIOQuantity[0] / 16) -496)));
				ITF_CLIENT_IN.DESTROY_JOB(_byMbFunction 		:= 16,	_wMbAdress 	:=24936,	_pData 	:=	 ADR(_ayAnalogOutput[616]),	_wQuantity	 :=	 MAX(1,MIN(120,(_ayIOQuantity[0] / 16) -616)));
				ITF_CLIENT_IN.DESTROY_JOB(_byMbFunction 		:= 16,	_wMbAdress 	:=25056,	_pData 	:=	 ADR(_ayAnalogOutput[736]),	_wQuantity	 :=	 MAX(1,MIN(120,(_ayIOQuantity[0] / 16) -736)));
				ITF_CLIENT_IN.DESTROY_JOB(_byMbFunction 		:= 16,	_wMbAdress 	:=25176,	_pData 	:=	 ADR(_ayAnalogOutput[856]),	_wQuantity	 :=	 MAX(1,MIN(120,(_ayIOQuantity[0] / 16) -856)));
				ITF_CLIENT_IN.DESTROY_JOB(_byMbFunction 		:= 16,	_wMbAdress 	:=25296,	_pData 	:=	 ADR(_ayAnalogOutput[976]),	_wQuantity	 :=	 MAX(1,MIN(044,(_ayIOQuantity[0] / 16) -976)));	
				
				(* Delete Read Digital Input Jobs *)                                                  	       	  	                                  	   	
				ITF_CLIENT_IN.DESTROY_JOB(_byMbFunction 		:= 02,	_wMbAdress 	:= 0000,	_pData 	:=	 ADR(_ayDigitalInput[000]),	_wQuantity	 :=	 512);	
		
				(* Delete Read Digital Input Jobs *)                                                  	       	  	                                  	   	
				ITF_CLIENT_IN.DESTROY_JOB(_byMbFunction 		:= 15,	_wMbAdress 	:= 0000,	_pData 	:=	 ADR(_ayDigitalOutput[000]),_wQuantity	 :=	 512);		
			
				IF xReset THEN
					REM_ERROR();
					_wSoftWareReset := 16#AA55;
					ITF_CLIENT_IN.CREATE_JOB(_byMbFunction 		:= 06,	_wMbAdress 	:=8256,	_pData 	:=	 ADR(_wSoftWareReset),	_wQuantity	 :=	 1);	
					usiCase :=  usiCase + 1;
					xReset := FALSE;
					tErrorDelayMb := T#20S;   		// Neustart des FC Busüberwachung verlängern
				END_IF;
			12:	(* Wait *)
				IF ITF_CLIENT_IN.CONFIRM_ALL_JOBS_DONE THEN
					ITF_CLIENT_IN.DESTROY_JOB(_byMbFunction 	:= 06,	_wMbAdress 	:=8256,	_pData 	:=	 ADR(_wSoftWareReset),	_wQuantity	 :=	 1);
					(* Next Step *)
					usiCase := usiCase + 1;
				END_IF;			
			ELSE
				usiCase := 0;
		END_CASE;
	ELSE
		tErrorDelayMb := T#20S;
		xLockDown := TRUE;
		xBusError := TRUE;
	END_IF;
	(* Report*)
	actReport();
ELSE
	IF NOT GET_STATE_READY_TO_SET_CONFIG AND NOT CONFIG_DONE AND _INIT_DONE_SIMULATION THEN
		SET_STATE_READY_TO_SET_CONFIG := TRUE;
	ELSIF GET_STATE_READY_TO_SET_CONFIG AND NOT CONFIG_DONE THEN
		CONFIG_DONE := TRUE;
	END_IF
END_IF;

PROPERTY proVISU_DIA_NAME : STRING
GET
proVISU_DIA_NAME := 'CtaDevIOMb750362.DIA_MB750362';
END_GET
END_PROPERTY

ACTION actReport:
fbReportManager(stErrorInitReportTextListIn		:= ADR(GVL_TEXTLIST.stErrorTextlist),
				stWarningInitReportTextListIn	:= ADR(GVL_TEXTLIST.stWarningTextlist),
				stInfoInitReportTextListIn		:= ADR(GVL_TEXTLIST.stInfoTextlist),
				scReportNr						:= scReportNr);
				
(* Gett Quitt State *)
IF 	fbDevErrorReport.metGetQuitt() AND NOT xTrigResetSlotError  THEN
	xTrigResetSlotError	:= TRUE;
	xReset := TRUE;
ELSIF NOT fbDevErrorReport.metGetQuitt() THEN
	xTrigResetSlotError	:= FALSE;
END_IF;				

IF 	fbDevErrorReport.metGetQuitt() AND NOT xTrigResetDevError  THEN
	xTrigResetDevError	:= TRUE;
	xReset := TRUE;
ELSIF NOT fbDevErrorReport.metGetQuitt() THEN
	xTrigResetDevError	:= FALSE;
END_IF;		

fbMbErrorReport.metReport(xSetReportIn				:= xBusError,
						  iReportID					:= 1,
						  enReportTypeIn			:= CtaAppReport.enReportType.Error,
						  enReportAcknowledgeTypeIn	:= CtaAppReport.enReportacknowledgeType.Quit,
						  tDelay					:= tErrorDelayMb,
						  ITF_BMK_IN				:= THIS^,
						  pstReportTextListIn		:= ADR(GVL_TEXTLIST.stErrorTextlist),
						  stOptionalReportText		:= '',
						  iRetryTilReportLock		:= 0,
						  xResetCount				:= FALSE,
						  tReset					:= T#1S);
					
fbDevErrorReport.metReport(xSetReportIn				:= xLockDown,
						  iReportID					:= 2,
						  enReportTypeIn			:= CtaAppReport.enReportType.Error,
						  enReportAcknowledgeTypeIn	:= CtaAppReport.enReportacknowledgeType.Quit,
						  tDelay					:= T#1S,
						  ITF_BMK_IN				:= THIS^,
						  pstReportTextListIn		:= ADR(GVL_TEXTLIST.stErrorTextlist),
						  stOptionalReportText		:= '',
						  iRetryTilReportLock		:= 0,
						  xResetCount				:= FALSE,
						  tReset					:= T#1S);
						  
						  
fbWarningReportHand.metReport(	xSetReportIn				:= xHand,
						 	 	iReportID					:= 1,
						  		enReportTypeIn				:= CtaAppReport.enReportType.Warning,
						  		enReportAcknowledgeTypeIn	:= CtaAppReport.enReportacknowledgeType.Auto,
						 		tDelay						:= T#1S,
						  		ITF_BMK_IN					:= THIS^,
						  		pstReportTextListIn			:= ADR(GVL_TEXTLIST.stWarningTextlist),
						  		stOptionalReportText		:= '',
						  		iRetryTilReportLock			:= 0,
						  		xResetCount					:= FALSE,
						  		tReset						:= T#1S);

fbSlotMissmatch.metReport(xSetReportIn				:= xSlotMissmatch,
						  iReportID					:= 3,
						  enReportTypeIn			:= CtaAppReport.enReportType.Error,
						  enReportAcknowledgeTypeIn	:= CtaAppReport.enReportacknowledgeType.Quit,
						  tDelay					:= T#1S,
						  ITF_BMK_IN				:= THIS^,
						  pstReportTextListIn		:= ADR(GVL_TEXTLIST.stErrorTextlist),
						  stOptionalReportText		:= '',
						  iRetryTilReportLock		:= 0,
						  xResetCount				:= FALSE,
						  tReset					:= T#1S);
						  
						  
fbReportManager.metSyncReporter(fbMbErrorReport);
fbReportManager.metSyncReporter(fbDevErrorReport);
fbReportManager.metSyncReporter(fbWarningReportHand);
fbReportManager.metSyncReporter(fbSlotMissmatch);
END_ACTION

PROPERTY BUS_ERROR : BOOL
GET
BUS_ERROR := xBusError;
END_GET
END_PROPERTY

METHOD SIM_IO_TYPE
VAR_INPUT
	_usiSlotNr		: 	USINT;
	enSimIoTypeIn	:	CtaSysIO.enIOType;
	usiAnzIoType	:	USINT;
	_stSlotImage	:	STRING;
END_VAR
IF SIMULATION_ENABLED THEN
	_stSlotImage := fcGetModulImage(fcGetTypeOfWagoSlotSim(byAnzIo := usiAnzIoType,enSimIoTypeIn));
	SUPER^.SIM_IO_TYPE(_usiSlotNr,enSimIoTypeIn,usiAnzIoType,_stSlotImage);
END_IF;
END_METHOD

END_FUNCTION_BLOCK

// 30 Program Organization Units/FC/fcGetTypeOfWagoSlot
FUNCTION fcGetTypeOfWagoSlot : UINT
VAR_INPUT
	wInput	:	WORD;
END_VAR
VAR_OUTPUT
	xIsInput	:	BOOL;
	xIsDigital	:	BOOL;
	byAnzIo		:	BYTE;
	enModulType	:	enModuleType;
END_VAR

(* Check if its FCMB750362 *)
IF wInput = 362 THEN
	fcGetTypeOfWagoSlot := 362;
	xIsInput 			:= FALSE;
	byAnzIo				:= 0;
	enModulType			:= enModuleType.FCMB750362;	
ELSE
	(* Check if Digital Modul *)
	IF FcCheckIsDigitalIO(wIn := wInput,xIsInput => xIsInput , byAnzIo => byAnzIo) THEN
		xIsDigital := TRUE;
		(* Digital Input *)
		IF xIsInput THEN
			enModulType	:= enModuleType.Digital_IN;
			IF byAnzIo = 02 THEN
				fcGetTypeOfWagoSlot := 400; 	// 750-400
			ELSIF byAnzIo = 04 THEN
				fcGetTypeOfWagoSlot := 432; 	// 750-432		
			ELSIF byAnzIo = 08 THEN
				fcGetTypeOfWagoSlot := 1415; 	// 750-1415		
			ELSIF byAnzIo = 16 THEN
				fcGetTypeOfWagoSlot := 1405; 	// 750-1405				
			END_IF;
		(* Digital Output *)
		ELSE
			enModulType	:= enModuleType.Digital_OUT;
			IF byAnzIo = 02 THEN
				fcGetTypeOfWagoSlot := 501; 	// 750-501
			ELSIF byAnzIo = 04 THEN
				fcGetTypeOfWagoSlot := 515; 	// 750-515		
			ELSIF byAnzIo = 08 THEN
				fcGetTypeOfWagoSlot := 1515; 	// 750-1415		
			ELSIF byAnzIo = 16 THEN
				fcGetTypeOfWagoSlot := 1504; 	// 750-1504				
			END_IF;		
		END_IF;
	(* Analog or Spezial Modul *)
	ELSE
		IF wInput = 451 THEN
			fcGetTypeOfWagoSlot := 451;
			xIsInput 			:= TRUE;
			byAnzIo				:= 8;
			enModulType			:= enModuleType.TEMPERATUR;	
		ELSIF wInput = 455 THEN
			fcGetTypeOfWagoSlot := 455;
			xIsInput 			:= TRUE;
			byAnzIo				:= 4;
			enModulType			:= enModuleType.DC_4_20mA_IN;			
		ELSIF wInput = 459 THEN
			fcGetTypeOfWagoSlot := 459;
			xIsInput 			:= TRUE;
			byAnzIo				:= 4;
			enModulType			:= enModuleType.DC_0_10V_IN;			
		ELSIF wInput = 466 THEN
			fcGetTypeOfWagoSlot := 466;
			xIsInput 			:= TRUE;
			byAnzIo				:= 2;
			enModulType			:= enModuleType.DC_4_20mA_IN;			
		ELSIF wInput = 553 THEN 
			fcGetTypeOfWagoSlot := 553;
			xIsInput 			:= FALSE;
			byAnzIo				:= 4;
			enModulType			:= enModuleType.DC_0_20mA_OUT;	
		ELSIF wInput = 555 THEN
			fcGetTypeOfWagoSlot := 555;
			xIsInput 			:= FALSE;
			byAnzIo				:= 4;
			enModulType			:= enModuleType.DC_4_20mA_OUT;			
		ELSIF wInput = 597 THEN
			fcGetTypeOfWagoSlot := 597;
			xIsInput 			:= FALSE;
			byAnzIo				:= 8;
			enModulType			:= enModuleType.DC_0_10V_OUT;			
		ELSIF wInput = 652 THEN
			fcGetTypeOfWagoSlot := 652;
			xIsInput 			:= FALSE;
			byAnzIo				:= 48;
			enModulType			:= enModuleType.RS485;	
			{info '750-652 I/O must be Configuratet as 48byte via Wago I/O Check if used over Modbus'}		
		ELSIF wInput = 653 THEN
			fcGetTypeOfWagoSlot := 652;
			xIsInput 			:= FALSE;
			byAnzIo				:= 8;
			enModulType			:= enModuleType.RS485;			
		ELSE
			fcGetTypeOfWagoSlot := 0;
			xIsInput 			:= FALSE;
			byAnzIo				:= 0;
			enModulType			:= enModuleType.Unknown;			
		END_IF;
	END_IF;
END_IF;

END_FUNCTION

// 30 Program Organization Units/FC/FcCheckIsDigitalIO
FUNCTION FcCheckIsDigitalIO : BOOL
VAR_INPUT
	wIn			:	WORD;
END_VAR
VAR_OUTPUT
	xIsInput	:	BOOL;
	byAnzIo		:	BYTE;
END_VAR
VAR
END_VAR

FcCheckIsDigitalIO := wIn.15;
xIsInput 		   := wIn.0;
byAnzIo.0		   := wIn.8;
byAnzIo.1		   := wIn.9;
byAnzIo.2		   := wIn.10;
byAnzIo.3		   := wIn.11;
byAnzIo.4		   := wIn.12;
byAnzIo.5		   := wIn.13;
byAnzIo.6		   := wIn.14;

END_FUNCTION

// 30 Program Organization Units/FC/fcGetModulImage
FUNCTION fcGetModulImage : STRING
VAR_INPUT
	wIn			:	WORD;
END_VAR

VAR
    xIsInput    :   BOOL;
    byAnzIo   	:   BYTE;
END_VAR

(* END *)           
IF wIn = 600 THEN
	(* End Modul *)
	fcGetModulImage := '.WAGO_MB_IO_TERMINALS.0750_600';
ELSIF NOT FcCheckIsDigitalIO(wIn := wIn,xIsInput => xIsInput,byAnzIo => byAnzIo)  THEN  
	(* 750-451 *)
	IF wIn = 451 THEN
		fcGetModulImage := '.WAGO_MB_IO_TERMINALS.0750_451';    
	(* 750-455 *)
	ELSIF wIn = 455 THEN
		fcGetModulImage := '.WAGO_MB_IO_TERMINALS.0750_455';   
	(* 750-459 *)
	ELSIF wIn = 459 THEN
		fcGetModulImage := '.WAGO_MB_IO_TERMINALS.0750_459';   
	(* 750-466 *)
	ELSIF wIn = 466 THEN
		fcGetModulImage := '.WAGO_MB_IO_TERMINALS.0750_466';    
	(* 750-597 *)
	ELSIF wIn = 555 THEN
		fcGetModulImage := '.WAGO_MB_IO_TERMINALS.0750_555';   
	(* 750-597 *)
	ELSIF wIn = 597 THEN
		fcGetModulImage := '.WAGO_MB_IO_TERMINALS.0750_597';    
	(* 750-652 *)
	ELSIF wIn = 652 THEN
		fcGetModulImage := '.WAGO_MB_IO_TERMINALS.0750_652';     
	ELSE
	(* BLANK *)
		fcGetModulImage := '.WAGO_MB_IO_TERMINALS.0750_BLANK';      
	END_IF;
(* DI *)
ELSIF xIsInput THEN
	IF byAnzIo = 16 THEN
		(* 750-1405 *)
		fcGetModulImage := '.WAGO_MB_IO_TERMINALS.0750_1405';          
	ELSIF byAnzIo = 8 THEN
		(* 750-1415 *)
		fcGetModulImage := '.WAGO_MB_IO_TERMINALS.0750_1415';   
	ELSIF byAnzIo = 4 THEN
		(* 750-432 *)
		fcGetModulImage := '.WAGO_MB_IO_TERMINALS.0750_432';          
	ELSIF byAnzIo = 2 THEN
		(* 750-400 *)
		fcGetModulImage := '.WAGO_MB_IO_TERMINALS.0750_400';  
	ELSE
		(* 750-400 *)
		fcGetModulImage := '.WAGO_MB_IO_TERMINALS.0750_400';                                          
	END_IF;   
(* DO *)  
ELSIF NOT xIsInput THEN
	IF byAnzIo = 16 THEN
		(* 750-1504 *)
		fcGetModulImage := '.WAGO_MB_IO_TERMINALS.0750_1504'; 
	ELSE	
		(* 750-515 *)
		fcGetModulImage := '.WAGO_MB_IO_TERMINALS.0750_515';   
	END_IF; 
ELSE 
	(* Empty *)
	fcGetModulImage := '';
END_IF;

END_FUNCTION

// 30 Program Organization Units/FC/fcScaleIN0_10V
FUNCTION fcScaleIN0_10V : Real
VAR_INPUT
	wChanelInput	: WORD;	
END_VAR
VAR_OUTPUT
	xAlUnterlauf 	: BOOL;
	xAlUeberlauf	: BOOL;
END_VAR
VAR
	iChanelInput	: INT;
END_VAR

IF wChanelInput.0 = FALSE AND wChanelInput.1 = FALSE THEN
	// Für 12Bit Messwertausgabe die 3 Status Bit weglassen. Bit 15 kann vernachläsigt werden, da es immer 0 ist.
	iChanelInput 			:= WORD_TO_INT(SHR(wChanelInput,3)); 			// Prozesswert des AD Wandlers in INT										
	fcScaleIN0_10V			:= INT_TO_REAL(iChanelInput) /(4095.0/10.0);	// Skalierung des Messwertes auf 0-10V
// Störung: Sensorleitung ist Unterbrochen	
ELSIF wChanelInput.0 = TRUE	AND wChanelInput.1 = TRUE AND wChanelInput.2 = FALSE THEN
	xAlUnterlauf			:= TRUE;
    fcScaleIN0_10V			:= 0;
// Störung: Sensorleitung hat Überlauf	
ELSIF wChanelInput.0 = TRUE AND wChanelInput.1 = TRUE AND wChanelInput.2 = TRUE THEN
	xAlUeberlauf            := TRUE;
   	fcScaleIN0_10V          := 0;
END_IF

END_FUNCTION

// 30 Program Organization Units/FC/fcScaleIN4_20mA
FUNCTION fcScaleIN4_20mA : REAL
VAR_INPUT
	wChanelInput	: WORD; 
END_VAR	
VAR
	iChanelInput	: INT;	
END_VAR
VAR_OUTPUT
	xAlUeberlauf	: BOOL;
	xAlUnterlauf	: BOOL;
END_VAR

//  Prüfen der Error Bit 0 & Bit 1 
IF wChanelInput.0 = FALSE AND wChanelInput.1 = FALSE THEN
	// Für 12Bit Messwertausgabe die 3 Status Bit weglassen. Bit 15 kann vernachläsigt werden, da es immer 0 ist.
	iChanelInput 			:= WORD_TO_INT(SHR(wChanelInput,3)); 					// Prozesswert des AD Wandlers in INt										
	fcScaleIN4_20mA			:= INT_TO_REAL(iChanelInput) /(4095.0/16.0) + 4.0;		// Skalierung des Messwertes auf 4-20Ma
// Störung: Sensorleitung ist Unterbrochen	
ELSIF wChanelInput.0 = TRUE AND wChanelInput.1 = TRUE AND wChanelInput.2 = FALSE THEN 
    xAlUnterlauf        	:= TRUE;
    fcScaleIN4_20mA     	:= 0;
// Störung: Sensorleitung hat Überlauf	
ELSIF wChanelInput.0 = TRUE AND wChanelInput.1 = TRUE AND wChanelInput.2 = TRUE THEN
    xAlUeberlauf        	:= TRUE;
    fcScaleIN4_20mA     	:= 0;
END_IF;

END_FUNCTION

// 30 Program Organization Units/FC/fcScalePT1000
FUNCTION fcScalePT1000 : REAL
VAR_INPUT
	wChanelInput	: WORD;
END_VAR
VAR
	iChanelInput	: INT;	
END_VAR

VAR_OUTPUT
	xAlUeberlauf	: BOOL;
	xAlUnterlauf	: BOOL;
END_VAR

// Prüfen ob der Wert gültig ist
iChanelInput := TO_INT(wChanelInput);
IF iChanelInput > -2000 AND iChanelInput < 8500 THEN   
	// Temperaturausgabe
	fcScalePT1000		:= INT_TO_REAL(iChanelInput)/10.0;
// Störung: Sensorleitung ist Unterbrochen	
ELSIF iChanelInput >= 8500 THEN
    xAlUnterlauf        := TRUE;
    fcScalePT1000       := 1.0E-44;    
// Störung: Sensorleitung hat Kurzschluss	
ELSIF iChanelInput <= -2000  THEN 
    xAlUeberlauf        := TRUE;
    fcScalePT1000       := 3.402823E+38;   
END_IF;

END_FUNCTION

// 30 Program Organization Units/FC/fcScaleOut0_10V
FUNCTION fcScaleOut0_10V : WORD
VAR_INPUT
	rValueIn			: REAL;
END_VAR
VAR
	wMinCalcValue		: WORD;
	rPyhsicalMin		: REAL;
	rPysiclalMax		: REAL;
END_VAR

rPyhsicalMin		:= 0;
rPysiclalMax		:= 10;	
 
// Errechnung des minimalen Phyikalischen wertes
 wMinCalcValue   	:=  TO_WORD(TO_WORD(LIMIT(0,(rPyhsicalMin*((32767.0 - 0)/(rPysiclalMax-0)) + 0),32767)));
   
// Skalieren des Messwertes
fcScaleOut0_10V 	:=  TO_WORD(LIMIT(wMinCalcValue,(rValueIn - rPyhsicalMin)*((32767 - wMinCalcValue) / (rPysiclalMax-rPyhsicalMin))+ wMinCalcValue,32767));

END_FUNCTION

// 30 Program Organization Units/FC/fcScaleOut0_20mA
FUNCTION fcScaleOut0_20mA : WORD
VAR_INPUT
	rValueIn			: REAL;
END_VAR
VAR
	wMinCalcValue		: WORD;
	rPyhsicalMin		: REAL;
	rPysiclalMax		: REAL;
END_VAR

rPyhsicalMin		:= 0;
rPysiclalMax		:= 20;	
 
// Errechnung des minimalen Phyikalischen wertes
 wMinCalcValue   	:=  TO_WORD(TO_WORD(LIMIT(0,(rPyhsicalMin*((32767.0 - 0)/(rPysiclalMax-0)) + 0),32767)));
   
// Skalieren des Messwertes
fcScaleOut0_20mA 	:=  TO_WORD(LIMIT(wMinCalcValue,(rValueIn - rPyhsicalMin)*((32767 - wMinCalcValue) / (rPysiclalMax-rPyhsicalMin))+ wMinCalcValue,32767));

END_FUNCTION

// 30 Program Organization Units/FC/fcScaleOut4_20mA
FUNCTION fcScaleOut4_20mA : WORD
VAR_INPUT
	rValueIn			: REAL;
END_VAR
VAR
	wMinCalcValue		: WORD;
	rPyhsicalMin		: REAL;
	rPysiclalMax		: REAL;
END_VAR

rPyhsicalMin		:= 4;
rPysiclalMax		:= 20;	
 
// Errechnung des minimalen Phyikalischen wertes
 wMinCalcValue   	:=  TO_WORD(TO_WORD(LIMIT(0,(rPyhsicalMin*((32767.0 - 0)/(rPysiclalMax-0)) + 0),32767)));
   
// Skalieren des Messwertes
fcScaleOut4_20mA	:=  TO_WORD(LIMIT(wMinCalcValue,(rValueIn - rPyhsicalMin)*((32767 - wMinCalcValue) / (rPysiclalMax-rPyhsicalMin))+ wMinCalcValue,32767));

END_FUNCTION

// 30 Program Organization Units/FC/fcGetTypeOfWagoSlotSim
FUNCTION fcGetTypeOfWagoSlotSim : WORD
VAR_INPUT
	byAnzIo			:	BYTE;
	enSimIoTypeIn	:	CtaSysIO.enIOType;	
END_VAR

IF enSimIoTypeIn = CtaSysIO.enIOType.Digital_IN OR enSimIoTypeIn = CtaSysIO.enIOType.Digital_OUT THEN
	fcGetTypeOfWagoSlotSim := FcGetDigitalIOSim(byAnzIo,enSimIoTypeIn = CtaSysIO.enIOType.Digital_IN);
ELSE
	IF enSimIoTypeIn = CtaSysIO.enIOType.DC_0_10V_IN THEN
		IF byAnzIo = 4 THEN
			fcGetTypeOfWagoSlotSim := 459;
		ELSE
			fcGetTypeOfWagoSlotSim := 0;
		END_IF;	
	ELSIF enSimIoTypeIn = CtaSysIO.enIOType.DC_0_20mA_IN THEN
		fcGetTypeOfWagoSlotSim := 0;
	ELSIF enSimIoTypeIn = CtaSysIO.enIOType.DC_4_20mA_IN THEN
		IF byAnzIo = 2 THEN
			fcGetTypeOfWagoSlotSim := 466;
		ELSIF byAnzIo = 4 THEN
			fcGetTypeOfWagoSlotSim := 455;
		ELSE
			fcGetTypeOfWagoSlotSim := 0;
		END_IF;		
	ELSIF enSimIoTypeIn = CtaSysIO.enIOType.TEMPERATUR THEN
		IF byAnzIo = 8 THEN
			fcGetTypeOfWagoSlotSim := 451;
		ELSE
			fcGetTypeOfWagoSlotSim := 0;
		END_IF;		
	ELSIF enSimIoTypeIn = CtaSysIO.enIOType.DC_0_10V_OUT THEN
		IF byAnzIo = 8 THEN
			fcGetTypeOfWagoSlotSim := 597;
		ELSE
			fcGetTypeOfWagoSlotSim := 0;
		END_IF;				
	ELSIF enSimIoTypeIn = CtaSysIO.enIOType.DC_0_20mA_OUT THEN
		IF byAnzIo = 4 THEN
			fcGetTypeOfWagoSlotSim := 553;
		ELSE
			fcGetTypeOfWagoSlotSim := 0;
		END_IF;				
	ELSIF enSimIoTypeIn = CtaSysIO.enIOType.DC_4_20mA_OUT THEN
		IF byAnzIo = 4 THEN
			fcGetTypeOfWagoSlotSim := 555;
		ELSE
			fcGetTypeOfWagoSlotSim := 0;
		END_IF;		
	ELSE
		fcGetTypeOfWagoSlotSim := 0;		
	END_IF;
END_IF;

END_FUNCTION

// 30 Program Organization Units/FC/FcGetDigitalIOSim
FUNCTION FcGetDigitalIOSim : WORD
VAR_INPUT
	byAnzIo		:	BYTE;
	xIsInput	:	BOOL;
END_VAR

FcGetDigitalIOSim.15	:= TRUE;
FcGetDigitalIOSim.0	:= xIsInput ;
FcGetDigitalIOSim.8    := byAnzIo.0;
FcGetDigitalIOSim.9    := byAnzIo.1;
FcGetDigitalIOSim.10   := byAnzIo.2;
FcGetDigitalIOSim.11   := byAnzIo.3;
FcGetDigitalIOSim.12   := byAnzIo.4;
FcGetDigitalIOSim.13   := byAnzIo.5;
FcGetDigitalIOSim.14   := byAnzIo.6;

END_FUNCTION

// 30 Program Organization Units/FC/fcScaleIN0_20mA
FUNCTION fcScaleIN0_20mA : REAL
VAR_INPUT
	wChanelInput	: WORD; 
END_VAR	
VAR
	iChanelInput	: INT;	
END_VAR
VAR_OUTPUT
	xAlUeberlauf	: BOOL;
	xAlUnterlauf	: BOOL;
END_VAR

//  Prüfen der Error Bit 0 & Bit 1 
IF wChanelInput.0 = FALSE AND wChanelInput.1 = FALSE THEN
	// Für 12Bit Messwertausgabe die 3 Status Bit weglassen. Bit 15 kann vernachläsigt werden, da es immer 0 ist.
	iChanelInput 			:= WORD_TO_INT(SHR(wChanelInput,3)); 					// Prozesswert des AD Wandlers in INt										
	fcScaleIN0_20mA			:= INT_TO_REAL(iChanelInput) /(4095.0/20);				// Skalierung des Messwertes auf 0-20Ma
// Störung: Sensorleitung ist Unterbrochen	
ELSIF wChanelInput.0 = TRUE AND wChanelInput.1 = TRUE AND wChanelInput.2 = FALSE THEN 
    xAlUnterlauf        	:= TRUE;
    fcScaleIN0_20mA     	:= 0;
// Störung: Sensorleitung hat Überlauf	
ELSIF wChanelInput.0 = TRUE AND wChanelInput.1 = TRUE AND wChanelInput.2 = TRUE THEN
    xAlUeberlauf        	:= TRUE;
    fcScaleIN0_20mA     	:= 0;
END_IF;

END_FUNCTION

// 40 Visualizations/DIA_MB750362
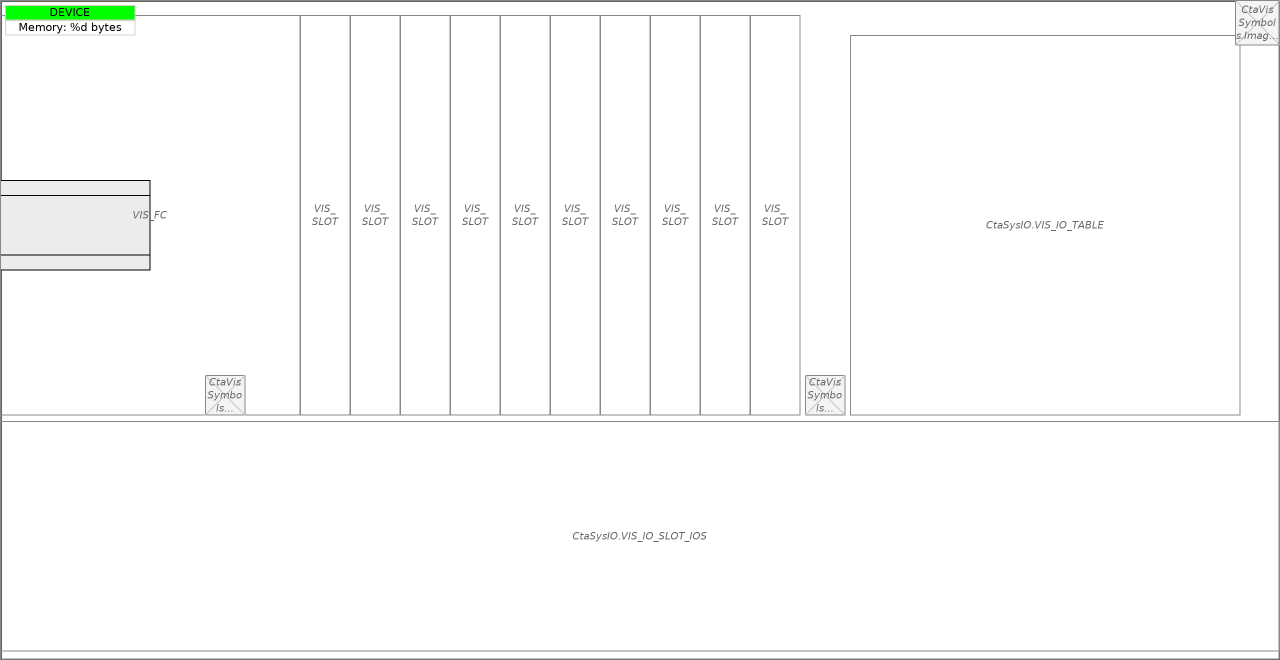
VISUALIZATION DIA_MB750362  // 1280x660
VAR_INPUT
	ITF_IO_DEVICE_IN : CtaSysIO.ITF_IO_DEVICE;
END_VAR
    Frame (0,0 1280x660), invisible if: NOT __QUERYINTERFACE(ITF_IO_DEVICE_IN,ITF_IO_DEVICE_IN)
        shows VIS_DYN_FC_IO_BASE(ITF_IO_DEVICE_IN := ITF_IO_DEVICE_IN)
    Image (1235,0 45x45), image: CtaVisSymbols.ImagePool.close_solo_black
        OnMouseClick:  Dialog=Current Dialog, Result=OK, NumpadKeypadSet=True
END_VISUALIZATION

// 40 Visualizations/PFC_SLOT/SLOT/VIS_SLOT
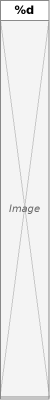
VISUALIZATION VIS_SLOT  // 50x400
VAR_INPUT
	ITF_IO_SLOT_IN :	CtaSysIO.ITF_IO_SLOT;
	xIsSelectet	   : 	BOOL;
END_VAR
    Frame (0,0 50x400), invisible if: NOT __QUERYINTERFACE(ITF_IO_SLOT_IN,ITF_IO_SLOT_IN)
        shows VIS_SLOT_QUERY(ITF_IO_SLOT_IN := ITF_IO_SLOT_IN, xIsSelectet := xIsSelectet)
END_VISUALIZATION

// 40 Visualizations/PFC_SLOT/SLOT/VIS_SLOT_QUERY
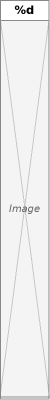
VISUALIZATION VIS_SLOT_QUERY  // 50x400
VAR_INPUT
	ITF_IO_SLOT_IN :	CtaSysIO.ITF_IO_SLOT;
	xIsSelectet	   : 	BOOL;
END_VAR
    Image (0,20 49x377), colour toggle: xIsSelectet
        p84334746: ITF_IO_SLOT_IN.IMAGE
    Textfield (0,0 49x20), "%d", text variable: ITF_IO_SLOT_IN.SLOT_NR
END_VISUALIZATION

// 40 Visualizations/PFC_SLOT/FC/VIS_FC
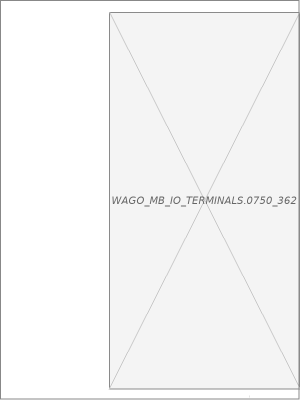
VISUALIZATION VIS_FC  // 300x400
VAR_INPUT
	ITF_IO_DEVICE_IN :	CtaSysIO.ITF_IO_DEVICE;
	ITF_IO_SLOT_IN :	CtaSysIO.ITF_IO_SLOT;
END_VAR
    Frame (0,0 300x400), invisible if: NOT __QUERYINTERFACE(ITF_IO_SLOT_IN,ITF_IO_SLOT_IN)
        shows VIS_FC_QUERY(ITF_IO_DEVICE_IN := ITF_IO_DEVICE_IN, ITF_IO_SLOT_IN := ITF_IO_SLOT_IN)
    Image (109,12 191x377), invisible if: __QUERYINTERFACE(ITF_IO_SLOT_IN,ITF_IO_SLOT_IN), image: WAGO_MB_IO_TERMINALS.0750_362
END_VISUALIZATION

// 40 Visualizations/PFC_SLOT/FC_SLOT
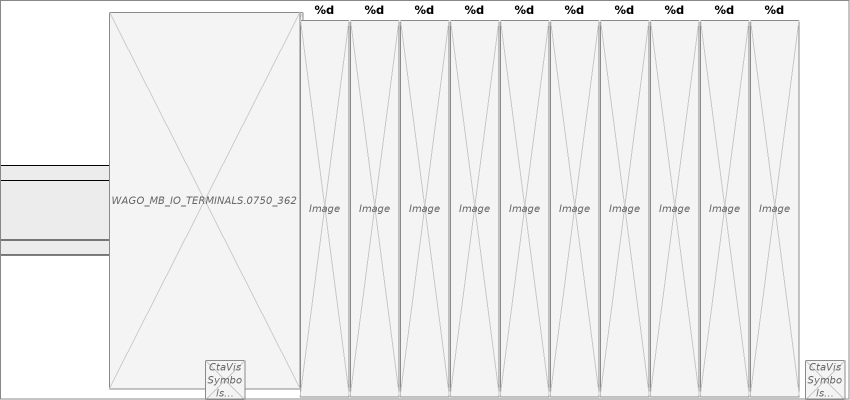
VISUALIZATION FC_SLOT  // 850x400
VAR_INPUT
	ITF_IO_DEVICE_IN :	CtaSysIO.ITF_IO_DEVICE;
END_VAR
VAR_IN_OUT
	ITF_IO_SLOT_IN	 :  CtaSysIO.ITF_IO_SLOT;
END_VAR
    Frame (0,0 850x400)
        shows FC_SLOT_QUERY(ITF_IO_DEVICE_IN := ITF_IO_DEVICE_IN, AY_ITF_SLOT := ITF_IO_DEVICE_IN.AY_ITF_SLOT_VIS, ITF_IO_SLOT_IN := ITF_IO_SLOT_IN)
END_VISUALIZATION

// 40 Visualizations/PFC_SLOT/FC_SLOT_QUERY
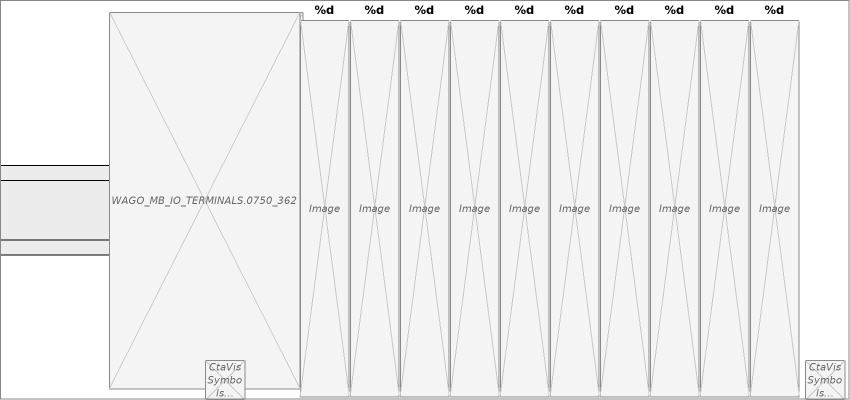
VISUALIZATION FC_SLOT_QUERY  // 850x400
VAR_INPUT
	ITF_IO_DEVICE_IN :	CtaSysIO.ITF_IO_DEVICE;
	AY_ITF_SLOT		 :	ARRAY[1..10] OF CtaSysIO.ITF_IO_SLOT;
END_VAR
VAR_IN_OUT
	ITF_IO_SLOT_IN	 :  CtaSysIO.ITF_IO_SLOT;
END_VAR
VAR
	usiSelectet		 :	USINT	:= 1;
END_VAR
    Group (0,165 803x90)
        Rectangle (0,0 150x90)
        Rectangle (0,15 150x60)
    Frame (0,0 300x400)
        shows VIS_FC(ITF_IO_DEVICE_IN := ITF_IO_DEVICE_IN, ITF_IO_SLOT_IN := AY_ITF_SLOT[1])
    Image (205,360 40x40), invisible if: SEL(__QUERYINTERFACE(AY_ITF_SLOT[1],AY_ITF_SLOT[1]),TRUE,AY_ITF_SLOT[1].SLOT_NR = 1), image: CtaVisSymbols.ImagePool.arrow-left_solo_black
        OnMouseClick: execute {
            ITF_IO_DEVICE_IN.RELOAD_ARRAY(FALSE,FALSE,TRUE);
            AY_ITF_SLOT := ITF_IO_DEVICE_IN.AY_ITF_SLOT_VIS;
            ITF_IO_SLOT_IN := AY_ITF_SLOT[1];
            usiSelectet	:= 1;
        }
    Image (805,360 40x40), invisible if: NOT __QUERYINTERFACE(AY_ITF_SLOT[10],AY_ITF_SLOT[10]), image: CtaVisSymbols.ImagePool.arrow-right_solo_black
        OnMouseClick: execute {
            ITF_IO_DEVICE_IN.RELOAD_ARRAY(FALSE,TRUE,FALSE);
            AY_ITF_SLOT := ITF_IO_DEVICE_IN.AY_ITF_SLOT_VIS;
            ITF_IO_SLOT_IN := AY_ITF_SLOT[1];
            usiSelectet	:= 1;
        }
    Frame (300,0 50x400)
        shows VIS_SLOT(ITF_IO_SLOT_IN := AY_ITF_SLOT[1], xIsSelectet := SEL(usiSelectet = 1,FALSE,__QUERYINTERFACE(AY_ITF_SLOT[1],ITF_IO_SLOT_IN)))
        OnMouseClick: execute { usiSelectet	:= 1; }
    Frame (350,0 50x400)
        shows VIS_SLOT(ITF_IO_SLOT_IN := AY_ITF_SLOT[2], xIsSelectet := SEL(usiSelectet = 2,FALSE,__QUERYINTERFACE(AY_ITF_SLOT[2],ITF_IO_SLOT_IN)))
        OnMouseClick: execute { usiSelectet	:= 2; }
    Frame (400,0 50x400)
        shows VIS_SLOT(ITF_IO_SLOT_IN := AY_ITF_SLOT[3], xIsSelectet := SEL(usiSelectet = 3,FALSE,__QUERYINTERFACE(AY_ITF_SLOT[3],ITF_IO_SLOT_IN)))
        OnMouseClick: execute { usiSelectet	:= 3; }
    Frame (450,0 50x400)
        shows VIS_SLOT(ITF_IO_SLOT_IN := AY_ITF_SLOT[4], xIsSelectet := SEL(usiSelectet = 4,FALSE,__QUERYINTERFACE(AY_ITF_SLOT[4],ITF_IO_SLOT_IN)))
        OnMouseClick: execute { usiSelectet	:= 4; }
    Frame (500,0 50x400)
        shows VIS_SLOT(ITF_IO_SLOT_IN := AY_ITF_SLOT[5], xIsSelectet := SEL(usiSelectet = 5,FALSE,__QUERYINTERFACE(AY_ITF_SLOT[5],ITF_IO_SLOT_IN)))
        OnMouseClick: execute { usiSelectet	:= 5; }
    Frame (550,0 50x400)
        shows VIS_SLOT(ITF_IO_SLOT_IN := AY_ITF_SLOT[6], xIsSelectet := SEL(usiSelectet = 6,FALSE,__QUERYINTERFACE(AY_ITF_SLOT[6],ITF_IO_SLOT_IN)))
        OnMouseClick: execute { usiSelectet	:= 6; }
    Frame (600,0 50x400)
        shows VIS_SLOT(ITF_IO_SLOT_IN := AY_ITF_SLOT[7], xIsSelectet := SEL(usiSelectet = 7,FALSE,__QUERYINTERFACE(AY_ITF_SLOT[7],ITF_IO_SLOT_IN)))
        OnMouseClick: execute { usiSelectet	:= 7; }
    Frame (650,0 50x400)
        shows VIS_SLOT(ITF_IO_SLOT_IN := AY_ITF_SLOT[8], xIsSelectet := SEL(usiSelectet = 8,FALSE,__QUERYINTERFACE(AY_ITF_SLOT[8],ITF_IO_SLOT_IN)))
        OnMouseClick: execute { usiSelectet	:= 8; }
    Frame (700,0 50x400)
        shows VIS_SLOT(ITF_IO_SLOT_IN := AY_ITF_SLOT[9], xIsSelectet := SEL(usiSelectet = 9,FALSE,__QUERYINTERFACE(AY_ITF_SLOT[9],ITF_IO_SLOT_IN)))
        OnMouseClick: execute { usiSelectet	:= 9; }
    Frame (750,0 50x400)
        shows VIS_SLOT(ITF_IO_SLOT_IN := AY_ITF_SLOT[10], xIsSelectet := SEL(usiSelectet = 10,FALSE,__QUERYINTERFACE(AY_ITF_SLOT[10],ITF_IO_SLOT_IN)))
        OnMouseClick: execute { usiSelectet	:= 10; }
END_VISUALIZATION

// 40 Visualizations/IO_ManagerBusInfo
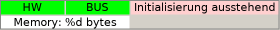
VISUALIZATION IO_ManagerBusInfo  // 280x30
VAR_INPUT
	xErrNotEnoughIOs	:	BOOL;
	xIoInitDone		    : 	BOOL;
	xKbusErrHW		    :	BOOL;
	xKbusErrSW		    : 	BOOL;
	udiNeededMemSize	: 	UDINT;
END_VAR
    Textfield (0,0 65x15), "HW Error", invisible if: NOT xKbusErrHW
    Textfield (0,0 65x15), "HW", invisible if: xKbusErrHW
    Textfield (65,0 65x15), "Reboot", invisible if: NOT xKbusErrSW
    Textfield (0,15 130x15), "Memory: %d bytes", text variable: udiNeededMemSize
    Textfield (130,0 150x15), "Initialisierung erfolgreich", invisible if: NOT xIoInitDone
    Textfield (130,0 150x15), "Initialisierung ausstehend", invisible if: xIoInitDone
    Textfield (65,0 65x15), "BUS", invisible if: xKbusErrSW
END_VISUALIZATION

// 40 Visualizations/VIS_DYN_FC_IO_BASE
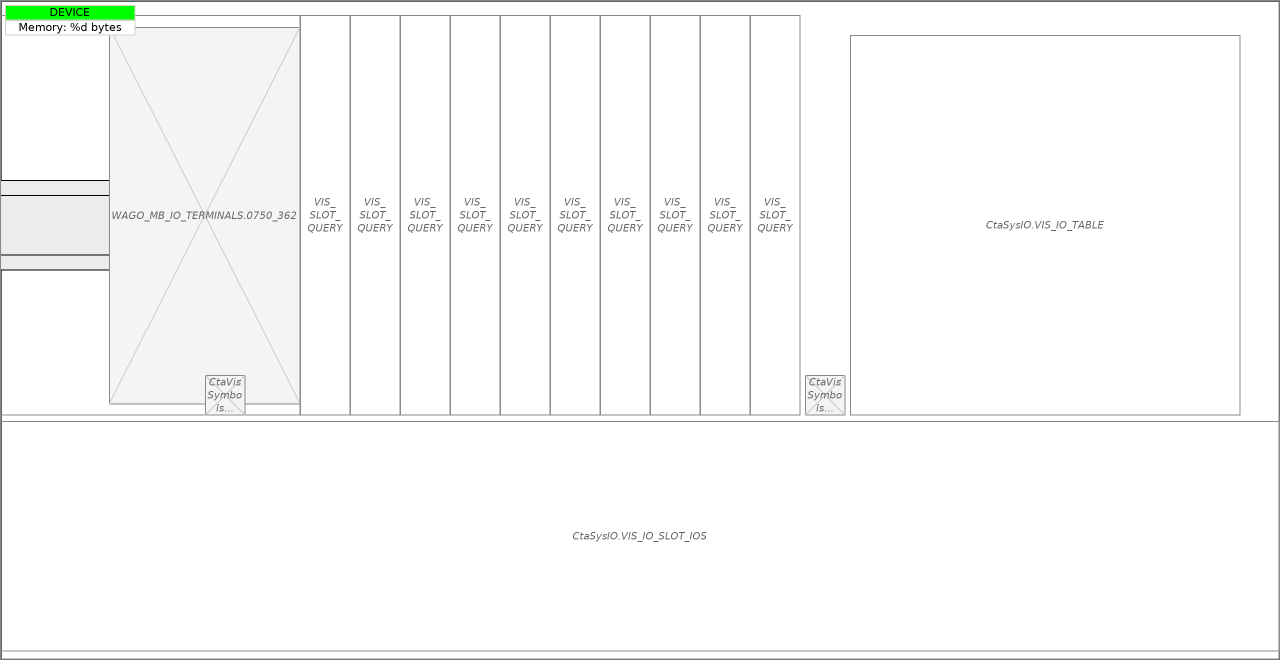
VISUALIZATION VIS_DYN_FC_IO_BASE  // 1280x660
VAR_INPUT
	ITF_IO_DEVICE_IN 	:	CtaSysIO.ITF_IO_DEVICE;
END_VAR
VAR
	ITF_IO_SLOT_TEMP	:	CtaSysIO.ITF_IO_SLOT;
END_VAR
    RoundedRectangle (0,0 1280x660)
    Frame (0,15 850x400), invisible if: NOT __QUERYINTERFACE(ITF_IO_DEVICE_IN,ITF_IO_DEVICE_IN)
        shows FC_SLOT(ITF_IO_DEVICE_IN := ITF_IO_DEVICE_IN, ITF_IO_SLOT_IN := ITF_IO_SLOT_TEMP)
    Frame (0,421 1280x230), invisible if: NOT __QUERYINTERFACE(ITF_IO_SLOT_TEMP,ITF_IO_SLOT_TEMP)
        shows CtaSysIO.VIS_IO_SLOT_IOS(ITF_IO_SLOT_IN := ITF_IO_SLOT_TEMP)
    Frame (850,35 390x380), invisible if: NOT __QUERYINTERFACE(ITF_IO_SLOT_TEMP,ITF_IO_SLOT_TEMP)
        shows CtaSysIO.VIS_IO_TABLE(ITF_IO_SLOT_IN := ITF_IO_SLOT_TEMP)
    Textfield (5,20 130x15), "Memory: %d bytes", text variable: ITF_IO_DEVICE_IN.DYN_SIZE
    Textfield (5,5 130x15), "DEVICE", colour toggle: ITF_IO_DEVICE_IN.ERROR
END_VISUALIZATION

// 40 Visualizations/PFC_SLOT/FC/VIS_FC_QUERY
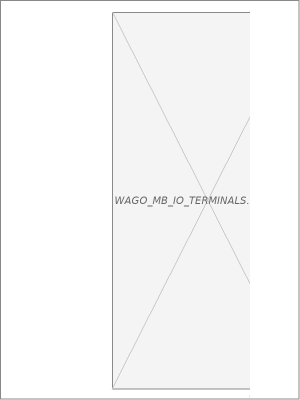
VISUALIZATION VIS_FC_QUERY  // 300x400
VAR_INPUT
	ITF_IO_DEVICE_IN :	CtaSysIO.ITF_IO_DEVICE;
	ITF_IO_SLOT_IN :	CtaSysIO.ITF_IO_SLOT;
END_VAR
    Image (112,12 191x377), invisible if: ITF_IO_SLOT_IN.SLOT_NR <> 1, image: WAGO_MB_IO_TERMINALS.0750_362
    Frame (250,0 50x400), invisible if: ITF_IO_SLOT_IN.SLOT_NR = 1
        shows VIS_SLOT(ITF_IO_SLOT_IN := ITF_IO_SLOT_IN.BIG_SYBIL, xIsSelectet := FALSE)
    Rectangle (250,0 50x400), invisible if: ITF_IO_SLOT_IN.SLOT_NR = 1
END_VISUALIZATION

(* text list txtModulType (id | default)
  Unknown | Unbekannt
  Digital_IN | Digital IN
  Digital_OUT | Digital OUT
  DC_0_10V_IN | DC 0-10V IN
  DC_0_10V_OUT | DC 0-10V OUT
  DC_4_20mA_IN | DC 4-20mA IN
  DC_4_20mA_OUT | DC 4-20mA Out
  ohm | Ohm
   |  *)

(* text list txtWarning (id | default)
  1 | IO Handeingriff
   |  *)

(* text list txtError (id | default)
  1 | Bus Kommunikations Fehler
  2 | FC750-362 Fehler
  3 | Slotkonfiguration nicht übereinstimmend
   |  *)

(* text list txtPhysicalUnit (id | default)
  0 | NaN
  1 | Digital In
  2 | Digital Out
  3 | 0 - 10 V
  4 | 4 - 20 mA
  5 | 0 - 10 V
  6 | 4 - 20 mA
  7 | °C
  8 | 
  9 | 0 - 20 mA
   |  *)

(* text list txtInfo (id | default)
   |  *)
